// SIMATIC S7-200 project (STEP 7-Micro/WIN), CPU 221 REL 01.10

ORGANIZATION_BLOCK MAIN:OB1
TITLE=PROGRAM COMMENTS  电动机顺序启停电路 
BEGIN
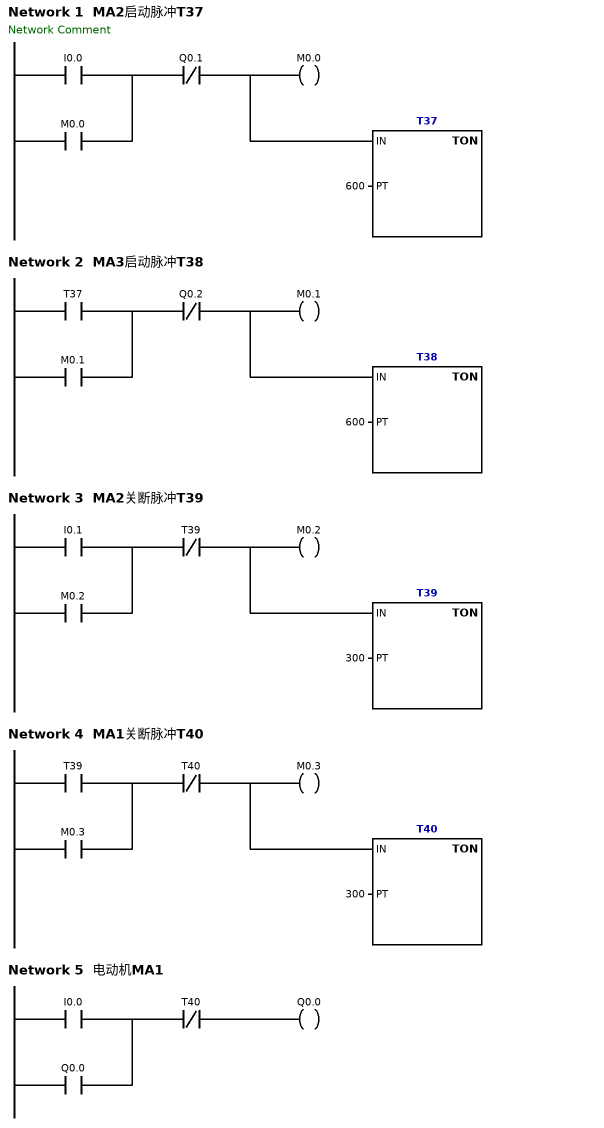
Network 1 // MA2启动脉冲T37
// Network Comment
LD     I0.0
O      M0.0
AN     Q0.1
=      M0.0
TON    T37, 600
Network 2 // MA3启动脉冲T38
LD     T37
O      M0.1
AN     Q0.2
=      M0.1
TON    T38, 600
Network 3 // MA2关断脉冲T39
LD     I0.1
O      M0.2
AN     T39
=      M0.2
TON    T39, 300
Network 4 // MA1关断脉冲T40
LD     T39
O      M0.3
AN     T40
=      M0.3
TON    T40, 300
Network 5 // 电动机MA1
LD     I0.0
O      Q0.0
AN     T40
=      Q0.0
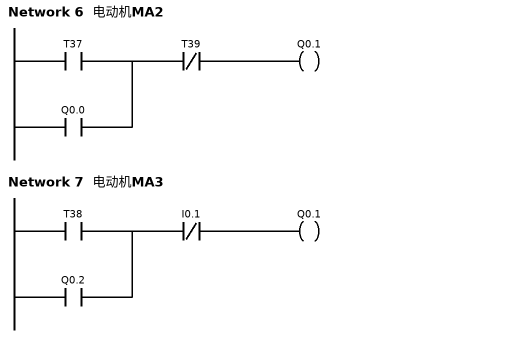
Network 6 // 电动机MA2
LD     T37
O      Q0.0
AN     T39
=      Q0.1
Network 7 // 电动机MA3
LD     T38
O      Q0.2
AN     I0.1
=      Q0.1
END_ORGANIZATION_BLOCK
